(* PLC project CoDeSys External Library Template, WAGO e!COCKPIT e!COCKPIT, author 3S - Smart Software Solutions GmbH *)
(* stored: creationDateTime 2019-10-29T12:37:19.8955215, version 3.5.5.30, modificationDateTime 2019-10-29T12:36:39.3744516, organization 3S - Smart Software Solutions GmbH *)
(* Library project template with all possible element types, docu and a sample project structure *)

FUNCTION fnKomunikatMACNadpisanie : STRING
  VAR_INPUT
    abMACAdres : ARRAY[1..6] OF BYTE;
  END_VAR
  VAR_IN_OUT
    sKomunikat : alSTRINGKomunikat;
  END_VAR
  VAR
    intBlad : INT;
    typKomunikat : typKomunikat;
  END_VAR

            

          
END_FUNCTION
